TYPE TFMachinePalletizer_WorkAreaZone :
STRUCT
	Zone		: ARRAY[1..MAXZONE] OF TFMachinePalletizer_Zone; (* Definizione Zone *)
END_STRUCT
END_TYPE

(* stored: Version 1.1.0.1, ProductVersion 3.1.4024.11
   DUT TFMachinePalletizer_WorkAreaZone: Id {68657dd1-bdbf-4e9d-a274-78a172a8dc38} *)
